// TIA Portal V20 export
FUNCTION_BLOCK "FB_AnalogInput"   // FB10, SCL
{ S7_Optimized_Access := 'FALSE' }
// stored: AutoNumber false, SetENOAutomatically false
   VAR_INPUT
      iValueHW { ExternalAccessible := 'False'; ExternalVisible := 'False'; ExternalWritable := 'False'} : Word;   // Value in word from PLC analog input
      iID : Int;
      iHMI_UpdateEnable : Bool;
   END_VAR
   VAR_IN_OUT
      ioAlarmOutOfRange { ExternalAccessible := 'False'; ExternalVisible := 'False'; ExternalWritable := 'False'} : Bool;   // Hardware signal out of nominal range alarm
      ioDataPLC : "AnalogInDataPLC_DT";
      ioDataHMI : "AnalogInDataHMI_DT";
      ioOPC : "UDT_OPC_Analog";
   END_VAR
   VAR
      sSWRealValue { ExternalAccessible := 'False'; ExternalVisible := 'False'; ExternalWritable := 'False'} : Real;
      sRT_Clock_1Hz : R_TRIG;
      sDownload { S7_SetPoint := 'True'} : Bool;   // Download DataHMI to OPC
   END_VAR
   VAR_TEMP
      tActual_input_value : Real;
   END_VAR
   VAR CONSTANT
      PT100 : UInt := 0;
      PT1000 : UInt := 1;
      TYP_0_10V : UInt := 2;
      "TYP_-10_10V" : UInt := 3;
      RES600 : UInt := 4;
      SL5201 : UInt := 5;
      PTC : UInt := 6;
   END_VAR
BEGIN
   REGION Description header 
       //==================================================================================
       // POSALUX Swiss SA / (C) Copyright 2025
       //----------------------------------------------------------------------------------
       // Title: AI_Alloc
       // Comment/Function:  Analog input management :  
       //                       - Based on input type (PT100, PT1000, 0-10V, -10+10V, RES600)  
       //                       - Value correction capability (y = Ax + B)  
       //                       - Alarm generation if measurement is out of tolerance (Alarm reset in FB_alarms)
       //                       - OPC Communication
       // Author: Fabien Waldt
       // Engineering: TIA Portal v17
       //----------------------------------------------------------------------------------
       // Change log table:
       // Version  | Date     | Expert in charge | Changes applied
       // ---------|----------|------------------|------------------------------------
       // 00.00.01 | 20250304 | FWA              | First released version
       // 00.00.02 | 20250610 | GSR              | Correction iAxFactor/iBOffset
       // 00.00.03 | 20251114 | FWA              | Add OPC Features
       // ==================================================================================
   END_REGION


   REGION Type of Probe
       CASE #ioDataPLC.TypeProbe OF
           #PT100:
               IF WORD_TO_INT(#iValueHW) <= 800 AND WORD_TO_INT(#iValueHW) >= -2000 THEN
                   #tActual_input_value := (INT_TO_REAL(WORD_TO_INT(#iValueHW)) * 0.1)*#ioDataHMI.AxFactor;
               ELSE
                   #tActual_input_value := 0.0;
                   #ioAlarmOutOfRange := TRUE;
               END_IF;

           #PT1000:
               IF WORD_TO_INT(#iValueHW) <= 800 AND WORD_TO_INT(#iValueHW) >= -2000 THEN
                   #tActual_input_value := (INT_TO_REAL(WORD_TO_INT(#iValueHW)) * 0.1)*#ioDataHMI.AxFactor;
               ELSE
                   #tActual_input_value := 0.0;
                   #ioAlarmOutOfRange := TRUE;
               END_IF;

           #TYP_0_10V:
               IF #iValueHW <= 27648 AND #iValueHW >= 0 THEN
                   #tActual_input_value := (((INT_TO_REAL(WORD_TO_INT(#iValueHW))*#ioDataHMI.AxFactor) * (#ioDataPLC.LimitUp - #ioDataPLC.LimitDown)) / 27648.0) *#ioDataHMI.AxFactor;
               ELSE
                   #tActual_input_value := 0.0;
                   #ioAlarmOutOfRange := TRUE;
               END_IF;

           #"TYP_-10_10V":
               IF (WORD_TO_INT(#iValueHW) <= 32767) AND (WORD_TO_INT(#iValueHW) >= -32767) THEN
                   #tActual_input_value := (((INT_TO_REAL(WORD_TO_INT(#iValueHW)) + 32767) * (#ioDataPLC.LimitUp - #ioDataPLC.LimitDown) / (2 * 32767))) *#ioDataHMI.AxFactor + #ioDataPLC.LimitDown;
               ELSE
                   #tActual_input_value := 0.0;
                   #ioAlarmOutOfRange := TRUE;
               END_IF;

           #RES600:
               IF #iValueHW <= 27648 AND #iValueHW >= 0 THEN
                   #tActual_input_value := (((INT_TO_REAL(WORD_TO_INT(#iValueHW))*#ioDataHMI.AxFactor) * (#ioDataPLC.LimitUp - #ioDataPLC.LimitDown)) / 27648.0) *#ioDataHMI.AxFactor ;
               ELSE
                   #tActual_input_value := 0.0;
                   #ioAlarmOutOfRange := TRUE;
               END_IF;
           #SL5201:
               IF #iValueHW <= 27648 AND #iValueHW >= 0 THEN
                   #tActual_input_value := (LREAL_TO_REAL(1.4774 * EXP(0.2536 * (WORD_TO_INT(#iValueHW) * 10.0 / 27648.0))))*#ioDataHMI.AxFactor;
               ELSE
                   #tActual_input_value := 0.0;
                   #ioAlarmOutOfRange := TRUE;
               END_IF;
           #PTC:
               IF #iValueHW.%X7 AND NOT #iValueHW.%X0 AND NOT #iValueHW.%X2 THEN
                   // Reaction to short-circuit : < 18 Ω -> SIMATIC S7: Bit 7 (IB x+1) = "1", Bit 0 = "0" and Bit 2 = "0"
                   // See documentation: Analog input module AI 4xRTD/TC 2-/3-/4-wire HF (6ES7134-6JD00-0CA1)
                   #ioAlarmOutOfRange := TRUE;
               ELSE
                   // No measurement value for PTC analog input ' bits 0 and 2 are handled in the related FB (Temperature)
                   // Normal range: < 550 Ω             -> Bit 0 = "0", Bit 2 = "0"
                   // Prewarning range: 550 Ω to 1650 Ω -> Bit 0 = "0", Bit 2 = "1"
                   // Response range: > 1650 Ω          -> Bit 0 = "1", Bit 2 = "0"
                   // See documentation Analog input module AI 4xRTD/TC 2-/3-/4-wire HF (6ES7134-6JD00-0CA1)
                   #tActual_input_value := (WORD_TO_INT(#iValueHW))*#ioDataHMI.AxFactor;
               END_IF;
       END_CASE;
   END_REGION

   REGION Update Values
       #sSWRealValue := #tActual_input_value + #ioDataHMI.BOffset;
       #ioDataHMI.CurrentValue := #sSWRealValue;
   END_REGION

   REGION OPC
       IF #ioOPC.Update AND #iHMI_UpdateEnable THEN
           // Copy HMI parameters (from OPC Parameters IHM) to HMI Datas (Used in PLC program)
           #ioDataHMI.StartTime := DINT_TO_TIME(REAL_TO_DINT(#ioOPC.Delay))*1000;
           #ioDataHMI.ThresholdAlarmMax := #ioOPC.DiffErrorMax;
           #ioDataHMI.ThresholdAlarmMin := #ioOPC.DiffErrorMin;
           #ioDataHMI.ThresholdWarningMax := #ioOPC.DiffWarnMax;
           #ioDataHMI.ThresholdWarningMin := #ioOPC.DiffWarnMin;
           #ioDataHMI.BOffset := #ioOPC.Offset;
           // #ioDataHMI.AxFactor := #ioOPC.Parameters.Gain; // Currently not on HMI
           #ioDataHMI.TargetValue := #ioOPC.Target;

           // Copy HMI Datas (Used in PLC program) to HMI (OPC Display HMI)
           #ioOPC.Delay := DINT_TO_REAL(TIME_TO_DINT(#ioDataHMI.StartTime)) / 1000.0;
           #ioOPC.DiffErrorMax := #ioDataHMI.ThresholdAlarmMax;
           #ioOPC.DiffErrorMin := #ioDataHMI.ThresholdAlarmMin;
           #ioOPC.DiffWarnMax := #ioDataHMI.ThresholdWarningMax;
           #ioOPC.DiffWarnMin := #ioDataHMI.ThresholdWarningMin;
           #ioOPC.Offset := #ioDataHMI.BOffset;
           // #ioOPC.Gain := #ioDataHMI.AxFactor; // Currently not on HMI
           #ioOPC.Target := #ioDataHMI.TargetValue;
           #ioOPC.Update := FALSE;
       END_IF;

       // Update ID
       #ioDataHMI.ID_Measure := #iID;
       #ioOPC.Id := #ioDataHMI.ID_Measure;

       // Update Current Value
       #sRT_Clock_1Hz(CLK := "Clock_1Hz");
       IF #sRT_Clock_1Hz.Q THEN
           #ioOPC.Value := #ioDataHMI.CurrentValue;
       END_IF;

       // Download DataHMI to OPC (Only used to initialize OPC Datas)
       IF #sDownload THEN
           // Copy HMI Datas (Used in PLC program) to HMI (OPC Display HMI)
           #ioOPC.Delay := DINT_TO_REAL(TIME_TO_DINT(#ioDataHMI.StartTime))/1000.0;
           #ioOPC.DiffErrorMax := #ioDataHMI.ThresholdAlarmMax;
           #ioOPC.DiffErrorMin := #ioDataHMI.ThresholdAlarmMin;
           #ioOPC.DiffWarnMax := #ioDataHMI.ThresholdWarningMax;
           #ioOPC.DiffWarnMin := #ioDataHMI.ThresholdWarningMin;
           #ioOPC.Offset := #ioDataHMI.BOffset;
           // #ioOPC.Gain := #ioDataHMI.AxFactor; // Currently not on HMI
           #ioOPC.Target := #ioDataHMI.TargetValue;
           #sDownload := FALSE;
       END_IF;
   END_REGION
END_FUNCTION_BLOCK
